{attribute 'GeneratedUsingTerminal: AX8108-0100-0101-0101'}
{attribute addProperty BoxType "AX8108-0100-0101-0101"}
{attribute addProperty Id "Ch_A_Position_actual_value_invalidAT %I*BOOL1Ch_A_1st_Additional_position_actual_value_invalidAT %I*BOOL1Ch_A_StatuswordAT %I*UINT2Ch_A_Position_actual_valueAT %I*DINT4"}
{attribute addProperty CRC "3692324381"}
{attribute addProperty Size "8"}
TYPE Ch_A_AxisMain_Inputs_DC14661D :
STRUCT
	{attribute addProperty Name "Ch_A_Position_actual_value_invalid"}
	Ch_A_Position_actual_value_invalid AT %I* : BOOL;
	{attribute addProperty Name "Ch_A_1st_Additional_position_actual_value_invalid"}
	Ch_A_1st_Additional_position_actual_value_invalid AT %I* : BOOL;
	{attribute addProperty Name "Ch_A_Statusword"}
	Ch_A_Statusword AT %I* : UINT;
	{attribute addProperty Name "Ch_A_Position_actual_value"}
	Ch_A_Position_actual_value AT %I* : DINT;
END_STRUCT
END_TYPE

(* stored: Version 1.2.0.0, ProductVersion 3.1.4024.9
   DUT Ch_A_AxisMain_Inputs_DC14661D: Id {3f3e3649-11d8-4540-8621-92bd07dada2a} *)
